// TIA Portal V17 export
// export: Created 2025-03-05T08:01:05.8765183Z, ExportSetting WithDefaults, DisplayName Totally Integrated Automation Portal, DisplayVersion V17 Update 8, DisplayName TIA Portal Openness, DisplayVersion V17 Update 8, DisplayName TIA Portal Version Control Interface, DisplayVersion V17, DisplayName SINAMICS Startdrive Advanced, DisplayVersion V17 SP2, DisplayName SINAMICS Startdrive G110M, G120, G120C, G120D, G120P, G115D, DisplayVersion V17 SP2, DisplayName SINAMICS Startdrive G130, G150, S120, S150, SINAMICS MV, S210, DisplayVersion V17 SP2, DisplayName STEP 7 Professional, DisplayVersion V17 Update 8, DisplayName SINUMERIK ONE STEP 7 Toolbox, DisplayVersion V17 Update 12, DisplayName SINUMERIK 840D sl STEP 7 Toolbox, DisplayVersion V17 Update 12, DisplayName STEP 7 Safety, DisplayVersion V17 Update 6, DisplayName WinCC Advanced, DisplayVersion V17 Update 8
DATA_BLOCK "DB1015_E-STOP"   // DB1015, F_DB
{ DB_Accessible_From_OPC_UA := 'FALSE' }
AUTHOR : ETXETAR
VERSION : 1.0
// stored: AutoNumber false, DBAccessibleFromOPCUA false, DBAccessibleFromWebserver true, InstanceOfName FB1015_E-STOP, InstanceOfType FB
"FB1015_E-STOP"
   // VAR_INPUT
   //    SAFETY_DOORS_BYPASS : Bool;
   //    FEEDBACK_OFF_E_STOP_IN : Bool;
   //    FEEDBACK_OFF_E_STOP_RST_STR_IN : Bool;
   //    MACH_E_STOP : Bool;
   //    GANTRY_E_STOP : Bool;
   //    POWDER_E_STOP : Bool;
   // END_VAR
   // VAR_OUTPUT
   //    E_STOP_OK : Bool;
   //    E_STOP_OK_OFF_DEL_2 : Bool;
   //    E_STOP_OK_OFF_DEL_3 : Bool;
   //    E_STOP_OK_OFF_DEL_4 : Bool;
   //    FEEDBACK_ERROR : Bool;
   // END_VAR
   // VAR
   //    ALL_E_STOP_IN : Bool;
   //    E_STOP_RESET : Bool;
   //    E_STOP_RESET_REQ : Bool;
   //    FEEDBACK_OFF_OK : Bool;
   //    ESTOP1_Instance : ESTOP1;
   //    F_IEC_Timer_Instance : TOF;
   //    F_IEC_Timer_Instance_1 : TOF;
   //    F_IEC_TIMER_FBCK_OK : TON;
   //    F_IEC_Timer_Instance_2 : TOF;
   // END_VAR
BEGIN
END_DATA_BLOCK
